{attribute addProperty BoxType "ELX3202-0000-0016"}
{attribute addProperty Id "RTD_Inputs_ChannelAT %I*ARRAY[0..1] OF RTD_Inputs_Channel_F16A160D6480WcStateAT %I*WcState_F855686C1620InfoDataAT %I*InfoData_BC63D37F80100"}
{attribute addProperty CRC "3045069298"}
{attribute addProperty SizeInBites "160"}
{attribute addProperty SizeInBytes "20"}
TYPE ELX3202_0EB9D2E9 :
STRUCT
	{attribute addProperty Name "RTD_Inputs_Channel"}
	RTD_Inputs_Channel : ARRAY[0..1] OF RTD_Inputs_Channel_F16A160D;
	{attribute addProperty Name "WcState"}
	WcState : WcState_F855686C;
	{attribute addProperty Name "InfoData"}
	InfoData : InfoData_BC63D37F;
END_STRUCT
END_TYPE

(* stored: Version 1.2.0.0, ProductVersion 3.1.4024.9
   DUT ELX3202_0EB9D2E9: Id {86a4145d-4459-4151-967d-7af36f757153} *)
